(*
SPDX-FileCopyrightText: © 2026 Oleksandr Tiutyk <trofimich@gmail.com>
SPDX-License-Identifier: MIT
License: https://opensource.org/license/mit
*)

(*!
<summary>Enumerates the current storage slots of a UniqueDataSet.</summary>
<description>
The source is borrowed and must outlive the cursor. Enumeration has no guaranteed ordering. Do not mutate the
source during traversal. Current is a borrowed view and must not be released or modified as an owning
descriptor; it is invalidated by cursor advancement/reset or source mutation. The caller owns and explicitly
releases a dynamically created cursor. MoveNext stops advancing at the end position of an unchanged source;
repeated exhausted calls return FALSE until Reset.
A null constructor source is diagnosed by traversal/current access, never by FB_init.
</description>
*)

{attribute 'no_explicit_call' := 'do not call this function block directly'}
{attribute 'enable_dynamic_creation'}
FUNCTION_BLOCK UniqueDataSetEnumerator EXTENDS TOF_Core.Object IMPLEMENTS TOF_Core.IEnumerator
VAR_STAT
	//! <summary>Class name shared by all instances of this function block.</summary>
	{attribute 'hide'} 
	_ClassName : STRING := __POUNAME();
END_VAR
VAR
	{attribute 'hide'} 
	_UniqueSet : IReadOnlyUniqueDataSet;
	{attribute 'hide'} 
	_CurrentIndex : DINT := -1;
	
	{attribute 'hide'} 
	_GenericValue : TOF_Core.GENERIC_VALUE;
END_VAR

(*!
<summary>Borrows the concrete cursor class name without transferring storage ownership.</summary>
*)
{attribute 'monitoring' := 'call'}
PROPERTY ClassName : REFERENCE TO STRING
GET
ClassName REF= _ClassName;
END_GET
END_PROPERTY

(*!
<summary>Exposes a read-only borrowed view of the current entry.</summary>
<description>
Reading Current before the first successful MoveNext, after Reset or after exhaustion yields an empty
descriptor. Otherwise payload is borrowed, with no disposal rights. Do not modify or release the descriptor.
The view may change on subsequent property access, cursor movement or source mutation.
Missing source raises DataMemberNotSpecifiedException before source access or cursor advancement.
</description>
*)
{attribute 'monitoring' := 'call'}
PROPERTY FINAL Current : REFERENCE TO TOF_Core.GENERIC_VALUE
GET
requireSource();

IF _CurrentIndex >= 0 AND_THEN _CurrentIndex < _UniqueSet.Length THEN
	_GenericValue := _UniqueSet.GetByIndex(index := _CurrentIndex); 
ELSE
	_GenericValue.Reset();	
END_IF 

Current REF= _GenericValue;
END_GET
END_PROPERTY

(*!
<summary>Binds the borrowed source for enumeration.</summary>
<description>
The source must be non-null and outlive the cursor. Only the reference is assigned; no allocation, callbacks
or throwing validation are performed. A null source remains invalid configuration and is reported by
MoveNext or current-value access without throwing from initialization.
</description>
*)
METHOD FB_init : BOOL
VAR_INPUT
	bInitRetains : BOOL; // TRUE: the retain variables are initialized (reset warm / reset cold)
	bInCopyCode : BOOL;  // TRUE: the instance will be copied to the copy code afterward (online change)
	uniqueSet : IReadOnlyUniqueDataSet;
END_VAR
_UniqueSet := uniqueSet;
END_METHOD

(*!
<summary>Advances the cursor to the next source position.</summary>
<description>
The source must be live, non-null and structurally unchanged during traversal. TRUE identifies a current
entry. The index advances only while below source Length and stops at the end position. Repeated exhausted
calls return FALSE without incrementing the index; reading Current yields an empty descriptor. Reset allows
traversal from the beginning again. No snapshot or mutation detection is provided. Descendants cannot override
this cursor operation; advancement, reset and borrowed current views use the same cursor state.
Missing source raises DataMemberNotSpecifiedException before source access or cursor advancement.
</description>
*)
{attribute "object_name" := "MoveNext"}
METHOD FINAL MoveNext : BOOL
requireSource();

IF _CurrentIndex < _UniqueSet.Length THEN
	_CurrentIndex := _CurrentIndex + 1;
END_IF

MoveNext := _CurrentIndex < _UniqueSet.Length;
END_METHOD

(*!
<summary>Provides the library namespace for diagnostics.</summary>
<description>
Borrowed read-only reference to compiler-initialized metadata; no ownership transfer.
</description>
*)
{attribute 'monitoring' := 'call'}
PROPERTY NamespaceName : REFERENCE TO STRING
GET
NamespaceName REF= CurrentNamespace.Name;
END_GET
END_PROPERTY

(*!
<summary>Places the cursor before the first source entry.</summary>
<description>
The next MoveNext starts at zero. Does not modify the source or release payload; reading Current now yields an
empty descriptor. Descendants cannot override this cursor operation; advancement, reset and borrowed current
views use the same cursor state.
</description>
*)
{attribute "object_name" := "Reset"}
METHOD FINAL Reset
_CurrentIndex := -1;
END_METHOD

(*!
<summary>Reports the size of this function-block instance.</summary>
<description>
Measured in bytes; includes inline storage but excludes separately allocated buffers, payload and enumerators.
</description>
*)
{attribute 'monitoring' := 'call'}
PROPERTY SelfSize : ULINT
GET
SelfSize := XSIZEOF(THIS^);
END_GET
END_PROPERTY

(*!
<summary>Requires the configured source before traversal or current-value access.</summary>
<description>
A missing mandatory source is configuration failure, not an empty collection. Raises a framework diagnostic
outside lifecycle methods and before mutation; it does not validate arbitrary pointer lifetime.
</description>
*)
METHOD PRIVATE requireSource
IF _UniqueSet = 0 THEN
	TOF_Core.Exceptions.ThrowDataMemberNotSpecified(
		sourceNamespaceName := NamespaceName,
		sourceClassName := ClassName,
		sourcePOUName := __POUNAME(),
		sourcePosition := __POSITION(),
		dataMemberName := 'uniqueSet'
	);
END_IF
END_METHOD

END_FUNCTION_BLOCK

(* stored: Version 1.1.0.1
   POU UniqueDataSetEnumerator: Id {001fed71-03fc-49d4-9d27-7de735b3019f}, SpecialFunc None
   Property ClassName: Id {521e8ad5-8bad-4740-8400-2bedb9859780}
   Get Get: Id {3cf7aaaa-7df3-4f6f-a62d-3a1716d9139d}
   Property Current: Id {d38f885d-0998-415e-91ff-61034aff0340}
   Get Get: Id {4c061dfd-7be1-4571-8f29-3051480d9284}
   Method FB_init: Id {ebd26738-5b17-4a49-9140-115ac86ef6fa}
   Method MoveNext: Id {816d4a55-bb40-4e03-aba8-22aec6e0278b}
   Property NamespaceName: Id {7ad2fc19-6d48-49d2-ad0a-59f1e7348df7}
   Get Get: Id {8bc44e8f-9672-4d28-b4da-dc2fe31ee002}
   Method Reset: Id {34cf0439-5d01-4262-ac61-eef9d91b52bb}
   Property SelfSize: Id {43152015-3912-4e0b-b518-95b25241b15c}
   Get Get: Id {846d440b-35ba-4402-b6dd-377c53c8ef7e}
   Method requireSource: Id {6a456cbe-026b-4415-b06a-6b5f1ead9cc9} *)
